FUNCTION_BLOCK FB_WorkerDefGrid_Verify EXTENDS FB_WorkerDefGrid
VAR_OUTPUT
  bWateGateActive   AT%Q* : BOOL;     //  wate gate activation pulse
END_VAR
VAR
  lastEjected   : BOOL;   // stores state if last CT was ejected 
  tpEjectPulse  : TP := (PT:=T#100MS);
  
  // print manager reference
  _pPm : POINTER TO FB_ProdManager_DMAX;
END_VAR

METHOD PROTECTED  Attach : BOOL
VAR_INPUT
  iCT              : I_CT;                         (*container at triggered event position*)
END_VAR
VAR 
  bSuccess         : BOOL;
END_VAR
IF SUPER^.Attach(iCT:=iCT) THEN
  
  // do CT supervision here and decice what happens with this sheet
   bSuccess := TRUE;
  IF NOT iCT.bValid AND iCT.bProductPresent AND iCT.pJob <> 0 THEN
    bSuccess := FALSE;
    // tag for ejection
    iCT.pCT^.lPrOutput := EN_PrinterOutput.trash;
	END_IF

  // finish CT in production
  IF _pPm <> 0 THEN 
    _pPm^.CT_Finish(sCT:=iCT, bSuccess:=bSuccess);
  ELSE
    LogError('PrintManager not set');
	END_IF
  
  // select output
  IF iCT.pCT^.lPrOutput = EN_PrinterOutput.trash THEN
    // create eject trigger
    tpEjectPulse(IN:=TRUE);
    lastEjected := TRUE;
  ELSE
    tpEjectPulse(IN:=FALSE);
    lastEjected := FALSE;
	END_IF
  
END_IF
END_METHOD

(*
  Set PrintManager.
*)
METHOD InitWorkerVerify : BOOL
VAR_INPUT
  pPm : POINTER TO FB_ProdManager_DMAX;
END_VAR
IF pPm = 0 THEN LogError('Invalid Pm given'); END_IF

_pPm := pPm;  // register print manager reference
END_METHOD

METHOD   mJobStart
VAR_INPUT
	sJobDef	: CalmarCompPrint.I_JobDefinition;
END_VAR
END_METHOD

METHOD  mJobStop
VAR_INPUT
	sStatus	: CalmarCompPrint.I_JobStatus;
END_VAR
END_METHOD

METHOD Release : BOOL
VAR_INPUT
  iCT              : I_CT;                         (*container at triggered event position*)
END_VAR
IF SUPER^.Release(iCT := iCT) THEN
  ;
END_IF
END_METHOD

METHOD  work
VAR_INST
  fT_Pulse  : F_TRIG;
END_VAR
SUPER^.work();

IF _pAttachedCt <> 0 THEN
  tpEjectPulse(Q=>bWateGateActive);
  fT_Pulse(CLK:=bWateGateActive);
  
  // release
  IF tpEjectPulse.IN THEN
    IF fT_Pulse.Q THEN  
      tpEjectPulse(IN:=FALSE);
      LogLvl(Lvl:=E_LogSeverity.Debug, Msg:=F_Concat2('Eject CT: ', _pAttachedCt^.print(0)));
      Release(iCT:=_pAttachedCt^);
    END_IF
  ELSE
    Release(iCT:=_pAttachedCt^);
  END_IF
END_IF
END_METHOD

END_FUNCTION_BLOCK

(* stored: Version 1.1.0.1, ProductVersion 3.1.4024.11
   POU FB_WorkerDefGrid_Verify: Id {ba30a803-cb22-4c70-92de-a30f80d703f5}, SpecialFunc None
   Folder I_PrintStatusClient: Id {23849181-f341-4a97-883d-05a0394fe9c7}
   Method Attach: Id {ed09302e-2885-443a-873e-e5493c07daba}
   Method InitWorkerVerify: Id {b89f6ac4-9ac9-4bfe-8bb7-e25e99bfe006}
   Method mJobStart: Id {a3da76c1-e8dd-4ffa-be59-c4c0dd030a9a}
   Method mJobStop: Id {29b4b42c-fe9c-4710-b09b-abd55ea27d44}
   Method Release: Id {c5bbf20b-0ff6-499b-bfe5-090aa809106f}
   Method work: Id {f3293130-827d-4f71-beb2-d681c617967b} *)
